INTERFACE I_VisitSensors

METHOD VisitSensor
VAR_INPUT
	Sensor : I_Sensor;
END_VAR
END_METHOD

END_INTERFACE

(* stored: Version 1.1.0.1, ProductVersion 3.1.4024.12
   Itf I_VisitSensors: Id {8b247a8b-5b7e-4de6-8f4f-445f6f7b9eff}
   Method VisitSensor: Id {b400fa79-623e-4a75-b97a-ba492acee68f} *)
